# B&R Automation Studio project HMI_JARB
Automation Studio 4.8.2.72

## Configuration Config1

### Hardware
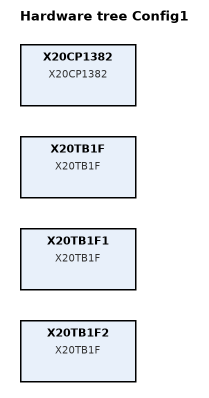
```
X20CP1382 : X20CP1382 v1.10.0.0  [X1 -> X1.SL; X2 -> X2.SL; X3 -> X3.SL]
  Module X1 (Type=X1, Virtual=true, Version=1.10.0.0)
    Connection (Connector=SS1, TargetModule=X20TB1F, TargetConnector=SS)
    Connection (Connector=SL, TargetModule=X20CP1382, TargetConnector=X1)
  Module X2 (Type=X2, Virtual=true, Version=1.10.0.0)
    Connection (Connector=SS1, TargetModule=X20TB1F1, TargetConnector=SS)
    Connection (Connector=SL, TargetModule=X20CP1382, TargetConnector=X2)
  Module X3 (Type=X3, Virtual=true, Version=1.10.0.0)
    Connection (Connector=SS1, TargetModule=X20TB1F2, TargetConnector=SS)
    Connection (Connector=SL, TargetModule=X20CP1382, TargetConnector=X3)
  Connector IF2:
    ActivateDevice = 1
    Vnc1
    VncVcObjectName1 = Visu
    VncKeyMappingFile1 = VC\PS2-Keyboard.dis
  ConfigurationID = HMI_JARB_Config1
  Simulation = 1
X20TB1F : X20TB1F v1.0.0.0
X20TB1F1 : X20TB1F v1.0.0.0
X20TB1F2 : X20TB1F v1.0.0.0
```

## Logical view

Binary libraries used (declarations not repeated): operator, runtime, astime, AsIecCon

### Library Logical/Libraries/Library (IEC)

#### Library.fun - Exported functions and function blocks
```iecst
{REDUND_ERROR} FUNCTION Addition : INT (* *) (*$GROUP=User,$CAT=User,$GROUPICON=User.png,$CATICON=User.png*)
	VAR_INPUT
		a : INT;
		b : INT;
	END_VAR
END_FUNCTION

{REDUND_ERROR} FUNCTION_BLOCK FUNKBLOK (*TODO: Add your comment here*) (*$GROUP=User,$CAT=User,$GROUPICON=User.png,$CATICON=User.png*)
	VAR_INPUT
		a : {REDUND_UNREPLICABLE} INT;
		b : {REDUND_UNREPLICABLE} INT;
	END_VAR
	VAR_OUTPUT
		Q : INT;
	END_VAR
	VAR RETAIN
		d : INT;
	END_VAR
END_FUNCTION_BLOCK
```

#### Addition.st
```iecst
(*  *)
FUNCTION Addition
	Addition := a + b;
END_FUNCTION
```

#### FUNKBLOK.st
```iecst
(* TODO: Add your comment here *)
FUNCTION_BLOCK FUNKBLOK
	Q := a + b;
	d := d + Q;
END_FUNCTION_BLOCK
```

### Program Logical/Program

#### Variables.var
```iecst
VAR
	c : INT;
	d : INT;
	FUNKBLOK2 : FUNKBLOK;
	out : INT;
END_VAR
```

#### Main.st
```iecst
PROGRAM _INIT
	(* Insert code here *)

END_PROGRAM

PROGRAM _CYCLIC
	(* Insert code here *)

	c := Addition(1,2);
	FUNKBLOK2(a:=1,b:=2);
	FUNKBLOK2.Q;

END_PROGRAM

PROGRAM _EXIT
	(* Insert code here *)

END_PROGRAM
```

Listed in the project but not available here: Logical/Libraries/Library/Types.typ, Logical/Libraries/Library/Constants.var
